# EPICS substitutions: ek9000App/Db/EL2084.substitutions
file EL2084.template
{       pattern
        {
                TERMINAL,

        }
        {
        }
}
